FUNCTION_BLOCK TransportSequenceBoot EXTENDS TransportSequence IMPLEMENTS ZCore.ISequence
VAR
  _step : ZCore.Step(TransportStep.BootBegin, TransportStep.BootEnd);
END_VAR

IF OnStart(_step) THEN
  ; // init custom sequence variables here ...
END_IF

REPEAT
  LogStep();

  CASE _step.Index OF
    (* -------------------------------------------------------------------------------------------------------------------------------- *)
    TransportStep.BootBegin:
    (* -------------------------------------------------------------------------------------------------------------------------------- *)
      IF _step.OnEntry()
      THEN
        // initialize equipment
        _io();
        _actuator();
        _fieldbus();
        _axis();
        _unit();
      END_IF
      
      _parent._objectManager.Cyclic();      
      Assert(_parent._objectManager);
      IF _parent._objectManager.Done
      THEN
        _step.SetNext(TransportStep.BootEnd);
      END_IF

    (* -------------------------------------------------------------------------------------------------------------------------------- *)
    TransportStep.BootEnd:
    (* -------------------------------------------------------------------------------------------------------------------------------- *)
      SetBusy(FALSE);
      
  ELSE
    Abort('sequence contains unhandled step');
  END_CASE
UNTIL _step.IsNotRepeatable() OR_ELSE NOT Busy END_REPEAT

END_FUNCTION_BLOCK

(* stored: Version 1.1.0.1
   POU TransportSequenceBoot: Id {52254bf8-b10a-40e1-8386-428d381258ff}, SpecialFunc None *)
